TYPE ST_DiscreteValveState :
STRUCT
	nPosition : E_DiscreteValvePosition;
END_STRUCT
END_TYPE

(* stored: Version 1.1.0.1, ProductVersion 3.1.4024.10
   DUT ST_DiscreteValveState: Id {05129783-53bd-4c22-88f0-65135c0932e7} *)
